TYPE csp_transfer_infeed_constant_accU :
STRUCT
	(*BELT Info*)
	MIN_VELOCITY_MMpSEC:						LREAL := 100;
	MAX_VELOCITY_MMpSEC:						LREAL := 666.5487;
	MAX_ACCELERATION_MMpSEC2:					LREAL := 6000;
	MAX_DECELERATION_MMpSEC2:					LREAL := 6000;
	MAX_JERK_MMpSEC3:							LREAL := 1000000;
	RUNNING_ACCELERATION_MMMpSEC2:				LREAL := 3000;
	RUNNING_DECELERATION_MMpSEC2:				LREAL := 3000;
	MAX_FOLLOWING_ERROR_MM:						LREAL := 100;
	
	RUNNING_JERK_MMpSEC3:						LREAL := 1000000;
	MOTOR_MAX_VELOCITY_DEGPS:					LREAL := 9600;
	MOTOR_MAX_ACCELERATION_DEGPS2:				LREAL := 4800;
	MOTOR_MAX_DECELERATION_DEGPS2:				LREAL := 4800;
	MOTOR_MAX_JERK_DEGPS3:						LREAL := 100000000; 
	MOTOR_MAX_FOLLOWING_ERROR_DEG:				LREAL := 2;
END_STRUCT
END_TYPE

(* stored: Version 1.1.0.1, ProductVersion 3.1.4024.3
   DUT csp_transfer_infeed_constant_accU: Id {466c165b-ffb9-4095-bcc1-502d23a20c57} *)
